Staubli VAL3: N18_TirarPuntes.pgx

program N18_TirarPuntes()
  local pointRx l_pTirarPuntes
begin

  // Anar al punt de tirar puntes
  l_pTirarPuntes=pTirarPuntes
  l_pTirarPuntes.trsf.x=l_pTirarPuntes.trsf.x+nXOffset
  l_pTirarPuntes.trsf.y=l_pTirarPuntes.trsf.y+nYOffset
  l_pTirarPuntes.trsf.z=l_pTirarPuntes.trsf.z+nZOffset
  movel(l_pTirarPuntes,tToolActiva,mLent)
  waitEndMove()

  bTaskDone=true
end
